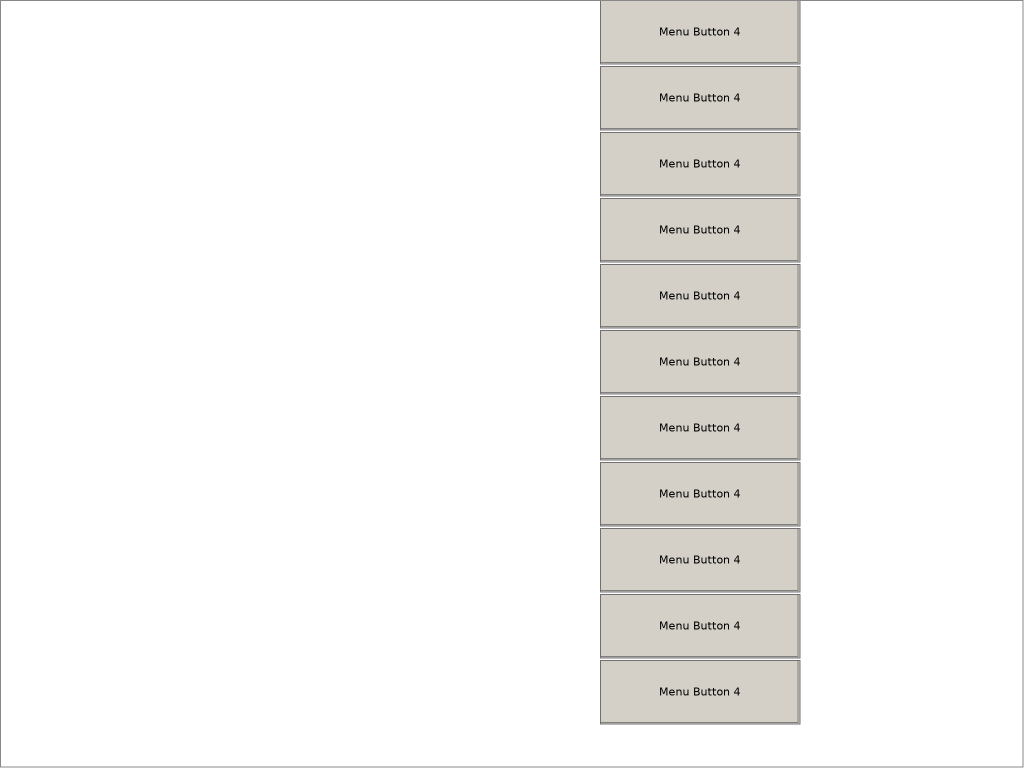
VISUALIZATION PopupMenu4  // 1024x768
    Button (600,0 200x64), "Menu Button 4"
        OnMouseClick: CloseDialog Dialog=PopupMenu4, Result=None, NumpadKeypadSet=True
    Button (600,66 200x64), "Menu Button 4"
        OnMouseClick: CloseDialog Dialog=PopupMenu4, Result=None, NumpadKeypadSet=True
    Button (600,132 200x64), "Menu Button 4"
        OnMouseClick: CloseDialog Dialog=PopupMenu4, Result=None, NumpadKeypadSet=True
    Button (600,198 200x64), "Menu Button 4"
        OnMouseClick: CloseDialog Dialog=PopupMenu4, Result=None, NumpadKeypadSet=True
    Button (600,264 200x64), "Menu Button 4"
        OnMouseClick: CloseDialog Dialog=PopupMenu4, Result=None, NumpadKeypadSet=True
    Button (600,330 200x64), "Menu Button 4"
        OnMouseClick: CloseDialog Dialog=PopupMenu4, Result=None, NumpadKeypadSet=True
    Button (600,396 200x64), "Menu Button 4"
        OnMouseClick: CloseDialog Dialog=PopupMenu4, Result=None, NumpadKeypadSet=True
    Button (600,462 200x64), "Menu Button 4"
        OnMouseClick: CloseDialog Dialog=PopupMenu4, Result=None, NumpadKeypadSet=True
    Button (600,528 200x64), "Menu Button 4"
        OnMouseClick: CloseDialog Dialog=PopupMenu4, Result=None, NumpadKeypadSet=True
    Button (600,594 200x64), "Menu Button 4"
        OnMouseClick: CloseDialog Dialog=PopupMenu4, Result=None, NumpadKeypadSet=True
    Button (600,660 200x64), "Menu Button 4"
        OnMouseClick: CloseDialog Dialog=PopupMenu4, Result=None, NumpadKeypadSet=True
    InvisibleInput (800,0 227x768)
        OnMouseClick: CloseDialog Dialog=PopupMenu4, Result=OK, NumpadKeypadSet=True
    InvisibleInput (0,0 600x768)
        OnMouseClick: CloseDialog Dialog=PopupMenu4, Result=OK, NumpadKeypadSet=True
    InvisibleInput (600,725 203x44)
        OnMouseClick: CloseDialog Dialog=PopupMenu4, Result=OK, NumpadKeypadSet=True
END_VISUALIZATION

(* stored: Version 1.1.0.1, ProductVersion 3.1.4024.11
   Visu PopupMenu4: Id {d63ed8df-94ed-0416-2992-3417057f4b4d} *)
